TYPE U_MOVER_CTRL :
UNION
  stCtrl              : ARRAY[1..MAX_MOVER] OF ST_MOVER_CTRL;

  byCtrl    AT %I*    : ARRAY[1..MAX_MOVER] OF
                        ARRAY[1..SIZEOF(ST_MOVER_CTRL)] OF BYTE;
END_UNION
END_TYPE

(* stored: Version 1.1.0.1, ProductVersion 3.1.4026.12
   DUT U_MOVER_CTRL: Id {1f94a128-e719-443d-972a-08c41a9c6fd7} *)
